FUNCTION_BLOCK FB_Movement_Teach
VAR_INPUT
	bExecute : BOOL;
	aArrangedFrames : ARRAY[0..60] OF Frame;
END_VAR
VAR_OUTPUT
END_VAR
VAR
	caseswitch : (init, prepare, executemovement, end, error);
	
	initPGT : R_TRIG; // used to detect first invokation of FB, stands for initialising postive going transition
	fbMover : FB_HbotMovement;
	fbHome : FB_HbotHome;
	iFrameCount : INT := 0;
	bNextFrame : BOOL;
	
	// HMI controls
	bRunSequence : BOOL;
	bRepeat : BOOL;
	bAbort : BOOL;
	bEnableHmiButton : BOOL; // This is to enable the HMI Buttons like abort, run sequence, repear...
	bExit: BOOL;
END_VAR

initPGT(CLK := bExecute);
IF initPGT.Q THEN // if the FB just started running, set case to init case to HOME (safety)
	iFrameCount := 0;
	caseswitch := prepare;
	bAbort := FALSE;
	bExit := FALSE;
	bEnableHmiButton := TRUE;
END_IF

CASE caseswitch OF 
//	init:
//		fbHome(bExecute := TRUE, StepperA := GVL.StepperReferenceA, StepperB := GVL.StepperReferenceB,
//			limitSwitchX := GVL.LimitSwitchX, limitSwitchY := GVL.LimitSwitchY);
//		IF fbHome.bError THEN
//			caseswitch := error;
//		ELSIF fbHome.bDone THEN
//			fbHome(bExecute := FALSE, StepperA := GVL.StepperReferenceA, StepperB := GVL.StepperReferenceB,
//			limitSwitchX := GVL.LimitSwitchX, limitSwitchY := GVL.LimitSwitchY);
//			caseswitch := prepare;
//		END_IF
		
	prepare:
		fbMover( bExecute := FALSE, StepperA := GVL.StepperReferenceA, StepperB := GVL.StepperReferenceB); // stop all movement
		IF aArrangedFrames[iFrameCount].Name = '' THEN
			iFrameCount := 0;
			
		END_IF
		
		IF bAbort THEN
			bExit := TRUE;	
			bEnableHmiButton := FALSE;
		ELSIF NOT bAbort THEN		
			IF bRunSequence THEN
				IF iFrameCount = 0 AND NOT bNextFrame THEN
					caseswitch := executemovement;
				ELSE
					iFrameCount := iFrameCount + 1;
					caseswitch := executemovement;
				END_IF
			END_IF
		END_IF
		
	executemovement:
		fbMover(MovementMode := fbMover.MoveAbsolute,
				rLinearSpeed := 60,
				rCurrentX := HbotForwardKinematics.rCurrentX,
				rCurrentY := HbotForwardKinematics.rCurrentY,
				rDeltaX := aArrangedFrames[iFrameCount].X,
				rDeltaY := aArrangedFrames[iFrameCount].Y,
				bExecute := TRUE,
				StepperA := GVL.StepperReferenceA,
				StepperB := GVL.StepperReferenceB);
		IF fbMover.bError THEN
			caseswitch := error; //catch errors
		ELSIF fbMover.bDone THEN
			bNextFrame := TRUE;
			caseswitch := prepare; // if it is done, go to the prep switch case
		END_IF
		IF NOT bRepeat THEN
			bRunSequence := FALSE;
		END_IF
		
END_CASE

END_FUNCTION_BLOCK

(* stored: Version 1.1.0.1, ProductVersion 3.1.4024.12
   POU FB_Movement_Teach: Id {637589ce-1047-4a20-a031-578f2b5d5925}, SpecialFunc None *)
